INTERFACE I_DigitalOutput EXTENDS I_DigitalDevice

PROPERTY Out : BOOL
GET
END_GET
SET
END_SET
END_PROPERTY

END_INTERFACE

(* stored: Version 1.1.0.1, ProductVersion 3.1.4024.12
   Itf I_DigitalOutput: Id {4c0288cf-c6d2-4267-848e-f61772f5ef93}
   Property Out: Id {7323f3fc-552d-42ba-9f27-1a6fe40770cd}
   Get Get: Id {ece55978-30da-43ec-b487-3cb2e47d95fa}
   Set Set: Id {d920bee1-f861-4ab8-ab5b-ae1bd65317b8} *)
